ABB RAPID module: dengju.mod

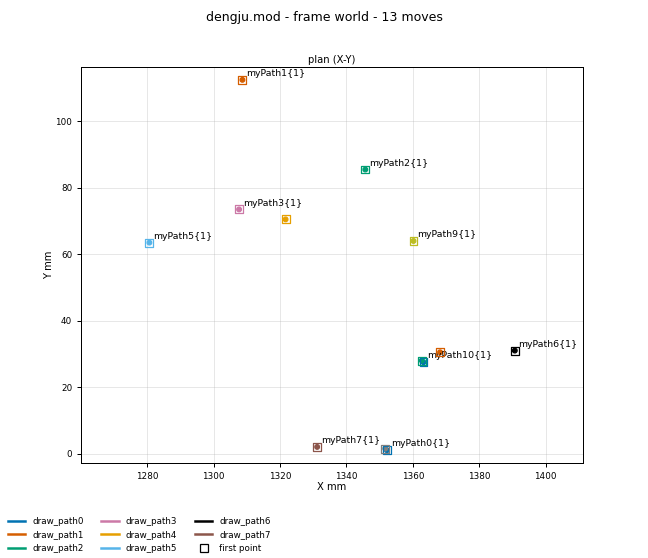
[picture p0: tool path of dengju.mod in frame world, 13 of 26 moves have a stored position in this frame; points joined in program order, loops and branches not executed]
MODULE Module1

    CONST robtarget myPath0{89} := [
        [[1352.2,1,938.01],[0.00139266,-0.491072,0.870802,-0.0234724],[0,-1,-1,0],[9E+09,9E+09,9E+09,9E+09,9E+09,9E+09]],
        [[1347.7,2.5,938.01],[0.00139266,-0.491072,0.870802,-0.0234724],[0,-1,-1,0],[9E+09,9E+09,9E+09,9E+09,9E+09,9E+09]],
        [[1342.2,4.5,938.01],[0.00139266,-0.491072,0.870802,-0.0234724],[0,-1,-1,0],[9E+09,9E+09,9E+09,9E+09,9E+09,9E+09]],
        [[1337.7,2,938.01],[0.00139266,-0.491072,0.870802,-0.0234724],[0,-1,-1,0],[9E+09,9E+09,9E+09,9E+09,9E+09,9E+09]],
        [[1331.7,1.5,938.01],[0.00139266,-0.491072,0.870802,-0.0234724],[0,-1,-1,0],[9E+09,9E+09,9E+09,9E+09,9E+09,9E+09]],
        [[1326.7,2.5,938.01],[0.00139266,-0.491072,0.870802,-0.0234724],[0,-1,-1,0],[9E+09,9E+09,9E+09,9E+09,9E+09,9E+09]],
        [[1322.2,4.5,938.01],[0.00139266,-0.491072,0.870802,-0.0234724],[0,-1,-1,0],[9E+09,9E+09,9E+09,9E+09,9E+09,9E+09]],
        [[1316.2,9.5,938.01],[0.00139266,-0.491072,0.870802,-0.0234724],[0,-1,-1,0],[9E+09,9E+09,9E+09,9E+09,9E+09,9E+09]],
        [[1311.2,14,938.01],[0.00139266,-0.491072,0.870802,-0.0234724],[0,-1,-1,0],[9E+09,9E+09,9E+09,9E+09,9E+09,9E+09]],
        [[1307.2,18,938.01],[0.00139266,-0.491072,0.870802,-0.0234724],[0,-1,-1,0],[9E+09,9E+09,9E+09,9E+09,9E+09,9E+09]],
        [[1304.2,22,938.01],[0.00139266,-0.491072,0.870802,-0.0234724],[0,-1,-1,0],[9E+09,9E+09,9E+09,9E+09,9E+09,9E+09]],
        [[1301.2,26,938.01],[0.00139266,-0.491072,0.870802,-0.0234724],[0,-1,-1,0],[9E+09,9E+09,9E+09,9E+09,9E+09,9E+09]],
        [[1298.7,30,938.01],[0.00139266,-0.491072,0.870802,-0.0234724],[0,-1,-1,0],[9E+09,9E+09,9E+09,9E+09,9E+09,9E+09]],
        [[1296.2,34,938.01],[0.00139266,-0.491072,0.870802,-0.0234724],[0,-1,-1,0],[9E+09,9E+09,9E+09,9E+09,9E+09,9E+09]],
        [[1294.2,38.5,938.01],[0.00139266,-0.491072,0.870802,-0.0234724],[0,-1,-1,0],[9E+09,9E+09,9E+09,9E+09,9E+09,9E+09]],
        [[1292.7,43,938.01],[0.00139266,-0.491072,0.870802,-0.0234724],[0,-1,-1,0],[9E+09,9E+09,9E+09,9E+09,9E+09,9E+09]],
        [[1291.7,51.5,938.01],[0.00139266,-0.491072,0.870802,-0.0234724],[0,-1,-1,0],[9E+09,9E+09,9E+09,9E+09,9E+09,9E+09]],
        [[1293.2,56.5,938.01],[0.00139266,-0.491072,0.870802,-0.0234724],[0,-1,-1,0],[9E+09,9E+09,9E+09,9E+09,9E+09,9E+09]],
        [[1296.7,62,938.01],[0.00139266,-0.491072,0.870802,-0.0234724],[0,-1,-1,0],[9E+09,9E+09,9E+09,9E+09,9E+09,9E+09]],
        [[1300.2,66,938.01],[0.00139266,-0.491072,0.870802,-0.0234724],[0,-1,-1,0],[9E+09,9E+09,9E+09,9E+09,9E+09,9E+09]],
        [[1304.7,69,938.01],[0.00139266,-0.491072,0.870802,-0.0234724],[0,-1,-1,0],[9E+09,9E+09,9E+09,9E+09,9E+09,9E+09]],
        [[1309.2,70.5,938.01],[0.00139266,-0.491072,0.870802,-0.0234724],[0,-1,-1,0],[9E+09,9E+09,9E+09,9E+09,9E+09,9E+09]],
        [[1314.2,71.5,938.01],[0.00139266,-0.491072,0.870802,-0.0234724],[0,-1,-1,0],[9E+09,9E+09,9E+09,9E+09,9E+09,9E+09]],
        [[1318.2,72,938.01],[0.00139266,-0.491072,0.870802,-0.0234724],[0,-1,-1,0],[9E+09,9E+09,9E+09,9E+09,9E+09,9E+09]],
        [[1308.2,73,938.01],[0.00139266,-0.491072,0.870802,-0.0234724],[0,-1,-1,0],[9E+09,9E+09,9E+09,9E+09,9E+09,9E+09]],
        [[1301.2,74,938.01],[0.00139266,-0.491072,0.870802,-0.0234724],[0,-1,-1,0],[9E+09,9E+09,9E+09,9E+09,9E+09,9E+09]],
        [[1296.7,75.5,938.01],[0.00139266,-0.491072,0.870802,-0.0234724],[0,-1,-1,0],[9E+09,9E+09,9E+09,9E+09,9E+09,9E+09]],
        [[1291.7,78,938.01],[0.00139266,-0.491072,0.870802,-0.0234724],[0,-1,-1,0],[9E+09,9E+09,9E+09,9E+09,9E+09,9E+09]],
        [[1287.2,80.5,938.01],[0.00139266,-0.491072,0.870802,-0.0234724],[0,-1,-1,0],[9E+09,9E+09,9E+09,9E+09,9E+09,9E+09]],
        [[1281.7,76.5,938.01],[0.00139266,-0.491072,0.870802,-0.0234724],[0,-1,-1,0],[9E+09,9E+09,9E+09,9E+09,9E+09,9E+09]],
        [[1280.7,69.5,938.01],[0.00139266,-0.491072,0.870802,-0.0234724],[0,-1,-1,0],[9E+09,9E+09,9E+09,9E+09,9E+09,9E+09]],
        [[1283.7,65,938.01],[0.00139266,-0.491072,0.870802,-0.0234724],[0,-1,-1,0],[9E+09,9E+09,9E+09,9E+09,9E+09,9E+09]],
        [[1284.2,63.5,938.01],[0.00139266,-0.491072,0.870802,-0.0234724],[0,-1,-1,0],[9E+09,9E+09,9E+09,9E+09,9E+09,9E+09]],
        [[1279.2,64,938.01],[0.00139266,-0.491072,0.870802,-0.0234724],[0,-1,-1,0],[9E+09,9E+09,9E+09,9E+09,9E+09,9E+09]],
        [[1274.2,66,938.01],[0.00139266,-0.491072,0.870802,-0.0234724],[0,-1,-1,0],[9E+09,9E+09,9E+09,9E+09,9E+09,9E+09]],
        [[1267.2,72,938.01],[0.00139266,-0.491072,0.870802,-0.0234724],[0,-1,-1,0],[9E+09,9E+09,9E+09,9E+09,9E+09,9E+09]],
        [[1265.2,82.5,938.01],[0.00139266,-0.491072,0.870802,-0.0234724],[0,-1,-1,0],[9E+09,9E+09,9E+09,9E+09,9E+09,9E+09]],
        [[1269.2,88,938.01],[0.00139266,-0.491072,0.870802,-0.0234724],[0,-1,-1,0],[9E+09,9E+09,9E+09,9E+09,9E+09,9E+09]],
        [[1274.7,89.5,938.01],[0.00139266,-0.491072,0.870802,-0.0234724],[0,-1,-1,0],[9E+09,9E+09,9E+09,9E+09,9E+09,9E+09]],
        [[1279.7,90.5,938.01],[0.00139266,-0.491072,0.870802,-0.0234724],[0,-1,-1,0],[9E+09,9E+09,9E+09,9E+09,9E+09,9E+09]],
        [[1278.2,98,938.01],[0.00139266,-0.491072,0.870802,-0.0234724],[0,-1,-1,0],[9E+09,9E+09,9E+09,9E+09,9E+09,9E+09]],
        [[1278.2,105.5,938.01],[0.00139266,-0.491072,0.870802,-0.0234724],[0,-1,-1,0],[9E+09,9E+09,9E+09,9E+09,9E+09,9E+09]],
        [[1280.2,110,938.01],[0.00139266,-0.491072,0.870802,-0.0234724],[0,-1,-1,0],[9E+09,9E+09,9E+09,9E+09,9E+09,9E+09]],
        [[1283.7,115.5,938.01],[0.00139266,-0.491072,0.870802,-0.0234724],[0,-1,-1,0],[9E+09,9E+09,9E+09,9E+09,9E+09,9E+09]],
        [[1287.7,119.5,938.01],[0.00139266,-0.491072,0.870802,-0.0234724],[0,-1,-1,0],[9E+09,9E+09,9E+09,9E+09,9E+09,9E+09]],
        [[1293.7,121.5,938.01],[0.00139266,-0.491072,0.870802,-0.0234724],[0,-1,-1,0],[9E+09,9E+09,9E+09,9E+09,9E+09,9E+09]],
        [[1301.2,121.5,938.01],[0.00139266,-0.491072,0.870802,-0.0234724],[0,-1,-1,0],[9E+09,9E+09,9E+09,9E+09,9E+09,9E+09]],
        [[1305.7,120,938.01],[0.00139266,-0.491072,0.870802,-0.0234724],[0,-1,-1,0],[9E+09,9E+09,9E+09,9E+09,9E+09,9E+09]],
        [[1310.7,119,938.01],[0.00139266,-0.491072,0.870802,-0.0234724],[0,-1,-1,0],[9E+09,9E+09,9E+09,9E+09,9E+09,9E+09]],
        [[1311.7,115,938.01],[0.00139266,-0.491072,0.870802,-0.0234724],[0,-1,-1,0],[9E+09,9E+09,9E+09,9E+09,9E+09,9E+09]],
        [[1320.2,114,938.01],[0.00139266,-0.491072,0.870802,-0.0234724],[0,-1,-1,0],[9E+09,9E+09,9E+09,9E+09,9E+09,9E+09]],
        [[1324.7,120,938.01],[0.00139266,-0.491072,0.870802,-0.0234724],[0,-1,-1,0],[9E+09,9E+09,9E+09,9E+09,9E+09,9E+09]],
        [[1331.7,121.5,938.01],[0.00139266,-0.491072,0.870802,-0.0234724],[0,-1,-1,0],[9E+09,9E+09,9E+09,9E+09,9E+09,9E+09]],
        [[1337.7,122,938.01],[0.00139266,-0.491072,0.870802,-0.0234724],[0,-1,-1,0],[9E+09,9E+09,9E+09,9E+09,9E+09,9E+09]],
        [[1342.7,121,938.01],[0.00139266,-0.491072,0.870802,-0.0234724],[0,-1,-1,0],[9E+09,9E+09,9E+09,9E+09,9E+09,9E+09]],
        [[1345.7,116,938.01],[0.00139266,-0.491072,0.870802,-0.0234724],[0,-1,-1,0],[9E+09,9E+09,9E+09,9E+09,9E+09,9E+09]],
        [[1346.7,113,938.01],[0.00139266,-0.491072,0.870802,-0.0234724],[0,-1,-1,0],[9E+09,9E+09,9E+09,9E+09,9E+09,9E+09]],
        [[1351.2,111.5,938.01],[0.00139266,-0.491072,0.870802,-0.0234724],[0,-1,-1,0],[9E+09,9E+09,9E+09,9E+09,9E+09,9E+09]],
        [[1356.7,108,938.01],[0.00139266,-0.491072,0.870802,-0.0234724],[0,-1,-1,0],[9E+09,9E+09,9E+09,9E+09,9E+09,9E+09]],
        [[1354.7,103.5,938.01],[0.00139266,-0.491072,0.870802,-0.0234724],[0,-1,-1,0],[9E+09,9E+09,9E+09,9E+09,9E+09,9E+09]],
        [[1352.7,99,938.01],[0.00139266,-0.491072,0.870802,-0.0234724],[0,-1,-1,0],[9E+09,9E+09,9E+09,9E+09,9E+09,9E+09]],
        [[1351.2,94,938.01],[0.00139266,-0.491072,0.870802,-0.0234724],[0,-1,-1,0],[9E+09,9E+09,9E+09,9E+09,9E+09,9E+09]],
        [[1352.2,89,938.01],[0.00139266,-0.491072,0.870802,-0.0234724],[0,-1,-1,0],[9E+09,9E+09,9E+09,9E+09,9E+09,9E+09]],
        [[1351.7,85,938.01],[0.00139266,-0.491072,0.870802,-0.0234724],[0,-1,-1,0],[9E+09,9E+09,9E+09,9E+09,9E+09,9E+09]],
        [[1354.2,80.5,938.01],[0.00139266,-0.491072,0.870802,-0.0234724],[0,-1,-1,0],[9E+09,9E+09,9E+09,9E+09,9E+09,9E+09]],
        [[1361.2,80,938.01],[0.00139266,-0.491072,0.870802,-0.0234724],[0,-1,-1,0],[9E+09,9E+09,9E+09,9E+09,9E+09,9E+09]],
        [[1366.2,79,938.01],[0.00139266,-0.491072,0.870802,-0.0234724],[0,-1,-1,0],[9E+09,9E+09,9E+09,9E+09,9E+09,9E+09]],
        [[1371.2,77.5,938.01],[0.00139266,-0.491072,0.870802,-0.0234724],[0,-1,-1,0],[9E+09,9E+09,9E+09,9E+09,9E+09,9E+09]],
        [[1375.7,75.5,938.01],[0.00139266,-0.491072,0.870802,-0.0234724],[0,-1,-1,0],[9E+09,9E+09,9E+09,9E+09,9E+09,9E+09]],
        [[1380.2,73.5,938.01],[0.00139266,-0.491072,0.870802,-0.0234724],[0,-1,-1,0],[9E+09,9E+09,9E+09,9E+09,9E+09,9E+09]],
        [[1384.2,71,938.01],[0.00139266,-0.491072,0.870802,-0.0234724],[0,-1,-1,0],[9E+09,9E+09,9E+09,9E+09,9E+09,9E+09]],
        [[1388.2,68.5,938.01],[0.00139266,-0.491072,0.870802,-0.0234724],[0,-1,-1,0],[9E+09,9E+09,9E+09,9E+09,9E+09,9E+09]],
        [[1393.2,63.5,938.01],[0.00139266,-0.491072,0.870802,-0.0234724],[0,-1,-1,0],[9E+09,9E+09,9E+09,9E+09,9E+09,9E+09]],
        [[1395.7,59,938.01],[0.00139266,-0.491072,0.870802,-0.0234724],[0,-1,-1,0],[9E+09,9E+09,9E+09,9E+09,9E+09,9E+09]],
        [[1398.2,55,938.01],[0.00139266,-0.491072,0.870802,-0.0234724],[0,-1,-1,0],[9E+09,9E+09,9E+09,9E+09,9E+09,9E+09]],
        [[1398.7,49.5,938.01],[0.00139266,-0.491072,0.870802,-0.0234724],[0,-1,-1,0],[9E+09,9E+09,9E+09,9E+09,9E+09,9E+09]],
        [[1397.7,44.5,938.01],[0.00139266,-0.491072,0.870802,-0.0234724],[0,-1,-1,0],[9E+09,9E+09,9E+09,9E+09,9E+09,9E+09]],
        [[1401.2,41.5,938.01],[0.00139266,-0.491072,0.870802,-0.0234724],[0,-1,-1,0],[9E+09,9E+09,9E+09,9E+09,9E+09,9E+09]],
        [[1401.7,36,938.01],[0.00139266,-0.491072,0.870802,-0.0234724],[0,-1,-1,0],[9E+09,9E+09,9E+09,9E+09,9E+09,9E+09]],
        [[1397.7,32,938.01],[0.00139266,-0.491072,0.870802,-0.0234724],[0,-1,-1,0],[9E+09,9E+09,9E+09,9E+09,9E+09,9E+09]],
        [[1392.7,31,938.01],[0.00139266,-0.491072,0.870802,-0.0234724],[0,-1,-1,0],[9E+09,9E+09,9E+09,9E+09,9E+09,9E+09]],
        [[1385.7,26,938.01],[0.00139266,-0.491072,0.870802,-0.0234724],[0,-1,-1,0],[9E+09,9E+09,9E+09,9E+09,9E+09,9E+09]],
        [[1382.7,22,938.01],[0.00139266,-0.491072,0.870802,-0.0234724],[0,-1,-1,0],[9E+09,9E+09,9E+09,9E+09,9E+09,9E+09]],
        [[1380.2,18,938.01],[0.00139266,-0.491072,0.870802,-0.0234724],[0,-1,-1,0],[9E+09,9E+09,9E+09,9E+09,9E+09,9E+09]],
        [[1375.7,12.5,938.01],[0.00139266,-0.491072,0.870802,-0.0234724],[0,-1,-1,0],[9E+09,9E+09,9E+09,9E+09,9E+09,9E+09]],
        [[1371.2,7.5,938.01],[0.00139266,-0.491072,0.870802,-0.0234724],[0,-1,-1,0],[9E+09,9E+09,9E+09,9E+09,9E+09,9E+09]],
        [[1367.2,5,938.01],[0.00139266,-0.491072,0.870802,-0.0234724],[0,-1,-1,0],[9E+09,9E+09,9E+09,9E+09,9E+09,9E+09]],
        [[1362.7,2.5,938.01],[0.00139266,-0.491072,0.870802,-0.0234724],[0,-1,-1,0],[9E+09,9E+09,9E+09,9E+09,9E+09,9E+09]],
        [[1357.7,1.5,938.01],[0.00139266,-0.491072,0.870802,-0.0234724],[0,-1,-1,0],[9E+09,9E+09,9E+09,9E+09,9E+09,9E+09]]
        ];
    CONST robtarget myPath1{4} := [
        [[1308.7,112.5,938.01],[0.00139266,-0.491072,0.870802,-0.0234724],[0,-1,-1,0],[9E+09,9E+09,9E+09,9E+09,9E+09,9E+09]],
        [[1312.2,115.5,938.01],[0.00139266,-0.491072,0.870802,-0.0234724],[0,-1,-1,0],[9E+09,9E+09,9E+09,9E+09,9E+09,9E+09]],
        [[1310.2,119,938.01],[0.00139266,-0.491072,0.870802,-0.0234724],[0,-1,-1,0],[9E+09,9E+09,9E+09,9E+09,9E+09,9E+09]],
        [[1306.2,116.5,938.01],[0.00139266,-0.491072,0.870802,-0.0234724],[0,-1,-1,0],[9E+09,9E+09,9E+09,9E+09,9E+09,9E+09]]
        ];
    CONST robtarget myPath2{5} := [
        [[1345.7,85.5,938.01],[0.00139266,-0.491072,0.870802,-0.0234724],[0,-1,-1,0],[9E+09,9E+09,9E+09,9E+09,9E+09,9E+09]],
        [[1350.7,86.5,938.01],[0.00139266,-0.491072,0.870802,-0.0234724],[0,-1,-1,0],[9E+09,9E+09,9E+09,9E+09,9E+09,9E+09]],
        [[1352.2,93,938.01],[0.00139266,-0.491072,0.870802,-0.0234724],[0,-1,-1,0],[9E+09,9E+09,9E+09,9E+09,9E+09,9E+09]],
        [[1348.2,95.5,938.01],[0.00139266,-0.491072,0.870802,-0.0234724],[0,-1,-1,0],[9E+09,9E+09,9E+09,9E+09,9E+09,9E+09]],
        [[1342.2,92.5,938.01],[0.00139266,-0.491072,0.870802,-0.0234724],[0,-1,-1,0],[9E+09,9E+09,9E+09,9E+09,9E+09,9E+09]]
        ];
    CONST robtarget myPath3{54} := [
        [[1307.7,73.5,938.01],[0.00139266,-0.491072,0.870802,-0.0234724],[0,-1,-1,0],[9E+09,9E+09,9E+09,9E+09,9E+09,9E+09]],
        [[1317.2,73,938.01],[0.00139266,-0.491072,0.870802,-0.0234724],[0,-1,-1,0],[9E+09,9E+09,9E+09,9E+09,9E+09,9E+09]],
        [[1319.7,77,938.01],[0.00139266,-0.491072,0.870802,-0.0234724],[0,-1,-1,0],[9E+09,9E+09,9E+09,9E+09,9E+09,9E+09]],
        [[1323.7,82,938.01],[0.00139266,-0.491072,0.870802,-0.0234724],[0,-1,-1,0],[9E+09,9E+09,9E+09,9E+09,9E+09,9E+09]],
        [[1327.7,84.5,938.01],[0.00139266,-0.491072,0.870802,-0.0234724],[0,-1,-1,0],[9E+09,9E+09,9E+09,9E+09,9E+09,9E+09]],
        [[1332.7,87,938.01],[0.00139266,-0.491072,0.870802,-0.0234724],[0,-1,-1,0],[9E+09,9E+09,9E+09,9E+09,9E+09,9E+09]],
        [[1337.2,88.5,938.01],[0.00139266,-0.491072,0.870802,-0.0234724],[0,-1,-1,0],[9E+09,9E+09,9E+09,9E+09,9E+09,9E+09]],
        [[1342.2,89.5,938.01],[0.00139266,-0.491072,0.870802,-0.0234724],[0,-1,-1,0],[9E+09,9E+09,9E+09,9E+09,9E+09,9E+09]],
        [[1344.7,95,938.01],[0.00139266,-0.491072,0.870802,-0.0234724],[0,-1,-1,0],[9E+09,9E+09,9E+09,9E+09,9E+09,9E+09]],
        [[1350.7,95,938.01],[0.00139266,-0.491072,0.870802,-0.0234724],[0,-1,-1,0],[9E+09,9E+09,9E+09,9E+09,9E+09,9E+09]],
        [[1352.7,101,938.01],[0.00139266,-0.491072,0.870802,-0.0234724],[0,-1,-1,0],[9E+09,9E+09,9E+09,9E+09,9E+09,9E+09]],
        [[1356.7,105.5,938.01],[0.00139266,-0.491072,0.870802,-0.0234724],[0,-1,-1,0],[9E+09,9E+09,9E+09,9E+09,9E+09,9E+09]],
        [[1354.2,110.5,938.01],[0.00139266,-0.491072,0.870802,-0.0234724],[0,-1,-1,0],[9E+09,9E+09,9E+09,9E+09,9E+09,9E+09]],
        [[1349.2,112,938.01],[0.00139266,-0.491072,0.870802,-0.0234724],[0,-1,-1,0],[9E+09,9E+09,9E+09,9E+09,9E+09,9E+09]],
        [[1344.7,113.5,938.01],[0.00139266,-0.491072,0.870802,-0.0234724],[0,-1,-1,0],[9E+09,9E+09,9E+09,9E+09,9E+09,9E+09]],
        [[1342.7,107.5,938.01],[0.00139266,-0.491072,0.870802,-0.0234724],[0,-1,-1,0],[9E+09,9E+09,9E+09,9E+09,9E+09,9E+09]],
        [[1343.7,103.5,938.01],[0.00139266,-0.491072,0.870802,-0.0234724],[0,-1,-1,0],[9E+09,9E+09,9E+09,9E+09,9E+09,9E+09]],
        [[1343.7,103.5,938.01],[0.00139266,-0.491072,0.870802,-0.0234724],[0,-1,-1,0],[9E+09,9E+09,9E+09,9E+09,9E+09,9E+09]],
        [[1340.2,101,938.01],[0.00139266,-0.491072,0.870802,-0.0234724],[0,-1,-1,0],[9E+09,9E+09,9E+09,9E+09,9E+09,9E+09]],
        [[1341.7,104,938.01],[0.00139266,-0.491072,0.870802,-0.0234724],[0,-1,-1,0],[9E+09,9E+09,9E+09,9E+09,9E+09,9E+09]],
        [[1342.7,111,938.01],[0.00139266,-0.491072,0.870802,-0.0234724],[0,-1,-1,0],[9E+09,9E+09,9E+09,9E+09,9E+09,9E+09]],
        [[1344.7,115,938.01],[0.00139266,-0.491072,0.870802,-0.0234724],[0,-1,-1,0],[9E+09,9E+09,9E+09,9E+09,9E+09,9E+09]],
        [[1343.7,120.5,938.01],[0.00139266,-0.491072,0.870802,-0.0234724],[0,-1,-1,0],[9E+09,9E+09,9E+09,9E+09,9E+09,9E+09]],
        [[1338.2,121.5,938.01],[0.00139266,-0.491072,0.870802,-0.0234724],[0,-1,-1,0],[9E+09,9E+09,9E+09,9E+09,9E+09,9E+09]],
        [[1332.2,122,938.01],[0.00139266,-0.491072,0.870802,-0.0234724],[0,-1,-1,0],[9E+09,9E+09,9E+09,9E+09,9E+09,9E+09]],
        [[1327.2,121,938.01],[0.00139266,-0.491072,0.870802,-0.0234724],[0,-1,-1,0],[9E+09,9E+09,9E+09,9E+09,9E+09,9E+09]],
        [[1323.2,118,938.01],[0.00139266,-0.491072,0.870802,-0.0234724],[0,-1,-1,0],[9E+09,9E+09,9E+09,9E+09,9E+09,9E+09]],
        [[1320.7,114,938.01],[0.00139266,-0.491072,0.870802,-0.0234724],[0,-1,-1,0],[9E+09,9E+09,9E+09,9E+09,9E+09,9E+09]],
        [[1320.2,113.5,938.01],[0.00139266,-0.491072,0.870802,-0.0234724],[0,-1,-1,0],[9E+09,9E+09,9E+09,9E+09,9E+09,9E+09]],
        [[1314.2,114,938.01],[0.00139266,-0.491072,0.870802,-0.0234724],[0,-1,-1,0],[9E+09,9E+09,9E+09,9E+09,9E+09,9E+09]],
        [[1309.7,112.5,938.01],[0.00139266,-0.491072,0.870802,-0.0234724],[0,-1,-1,0],[9E+09,9E+09,9E+09,9E+09,9E+09,9E+09]],
        [[1309.2,106,938.01],[0.00139266,-0.491072,0.870802,-0.0234724],[0,-1,-1,0],[9E+09,9E+09,9E+09,9E+09,9E+09,9E+09]],
        [[1309.2,101,938.01],[0.00139266,-0.491072,0.870802,-0.0234724],[0,-1,-1,0],[9E+09,9E+09,9E+09,9E+09,9E+09,9E+09]],
        [[1306.7,96,938.01],[0.00139266,-0.491072,0.870802,-0.0234724],[0,-1,-1,0],[9E+09,9E+09,9E+09,9E+09,9E+09,9E+09]],
        [[1308.2,98,938.01],[0.00139266,-0.491072,0.870802,-0.0234724],[0,-1,-1,0],[9E+09,9E+09,9E+09,9E+09,9E+09,9E+09]],
        [[1309.2,104,938.01],[0.00139266,-0.491072,0.870802,-0.0234724],[0,-1,-1,0],[9E+09,9E+09,9E+09,9E+09,9E+09,9E+09]],
        [[1309.2,109.5,938.01],[0.00139266,-0.491072,0.870802,-0.0234724],[0,-1,-1,0],[9E+09,9E+09,9E+09,9E+09,9E+09,9E+09]],
        [[1307.7,114,938.01],[0.00139266,-0.491072,0.870802,-0.0234724],[0,-1,-1,0],[9E+09,9E+09,9E+09,9E+09,9E+09,9E+09]],
        [[1306.2,119,938.01],[0.00139266,-0.491072,0.870802,-0.0234724],[0,-1,-1,0],[9E+09,9E+09,9E+09,9E+09,9E+09,9E+09]],
        [[1301.7,121,938.01],[0.00139266,-0.491072,0.870802,-0.0234724],[0,-1,-1,0],[9E+09,9E+09,9E+09,9E+09,9E+09,9E+09]],
        [[1294.2,122,938.01],[0.00139266,-0.491072,0.870802,-0.0234724],[0,-1,-1,0],[9E+09,9E+09,9E+09,9E+09,9E+09,9E+09]],
        [[1289.7,120.5,938.01],[0.00139266,-0.491072,0.870802,-0.0234724],[0,-1,-1,0],[9E+09,9E+09,9E+09,9E+09,9E+09,9E+09]],
        [[1285.7,117.5,938.01],[0.00139266,-0.491072,0.870802,-0.0234724],[0,-1,-1,0],[9E+09,9E+09,9E+09,9E+09,9E+09,9E+09]],
        [[1281.7,113.5,938.01],[0.00139266,-0.491072,0.870802,-0.0234724],[0,-1,-1,0],[9E+09,9E+09,9E+09,9E+09,9E+09,9E+09]],
        [[1279.7,109,938.01],[0.00139266,-0.491072,0.870802,-0.0234724],[0,-1,-1,0],[9E+09,9E+09,9E+09,9E+09,9E+09,9E+09]],
        [[1278.2,102.5,938.01],[0.00139266,-0.491072,0.870802,-0.0234724],[0,-1,-1,0],[9E+09,9E+09,9E+09,9E+09,9E+09,9E+09]],
        [[1278.2,94.5,938.01],[0.00139266,-0.491072,0.870802,-0.0234724],[0,-1,-1,0],[9E+09,9E+09,9E+09,9E+09,9E+09,9E+09]],
        [[1279.7,90,938.01],[0.00139266,-0.491072,0.870802,-0.0234724],[0,-1,-1,0],[9E+09,9E+09,9E+09,9E+09,9E+09,9E+09]],
        [[1282.2,86,938.01],[0.00139266,-0.491072,0.870802,-0.0234724],[0,-1,-1,0],[9E+09,9E+09,9E+09,9E+09,9E+09,9E+09]],
        [[1286.2,81.5,938.01],[0.00139266,-0.491072,0.870802,-0.0234724],[0,-1,-1,0],[9E+09,9E+09,9E+09,9E+09,9E+09,9E+09]],
        [[1290.2,78.5,938.01],[0.00139266,-0.491072,0.870802,-0.0234724],[0,-1,-1,0],[9E+09,9E+09,9E+09,9E+09,9E+09,9E+09]],
        [[1295.2,76,938.01],[0.00139266,-0.491072,0.870802,-0.0234724],[0,-1,-1,0],[9E+09,9E+09,9E+09,9E+09,9E+09,9E+09]],
        [[1299.7,74.5,938.01],[0.00139266,-0.491072,0.870802,-0.0234724],[0,-1,-1,0],[9E+09,9E+09,9E+09,9E+09,9E+09,9E+09]],
        [[1304.7,73.5,938.01],[0.00139266,-0.491072,0.870802,-0.0234724],[0,-1,-1,0],[9E+09,9E+09,9E+09,9E+09,9E+09,9E+09]]
        ];
    CONST robtarget myPath4{15} := [
        [[1321.7,70.5,938.01],[0.00139266,-0.491072,0.870802,-0.0234724],[0,-1,-1,0],[9E+09,9E+09,9E+09,9E+09,9E+09,9E+09]],
        [[1328.7,75,938.01],[0.00139266,-0.491072,0.870802,-0.0234724],[0,-1,-1,0],[9E+09,9E+09,9E+09,9E+09,9E+09,9E+09]],
        [[1333.2,77.5,938.01],[0.00139266,-0.491072,0.870802,-0.0234724],[0,-1,-1,0],[9E+09,9E+09,9E+09,9E+09,9E+09,9E+09]],
        [[1338.2,79,938.01],[0.00139266,-0.491072,0.870802,-0.0234724],[0,-1,-1,0],[9E+09,9E+09,9E+09,9E+09,9E+09,9E+09]],
        [[1343.7,80,938.01],[0.00139266,-0.491072,0.870802,-0.0234724],[0,-1,-1,0],[9E+09,9E+09,9E+09,9E+09,9E+09,9E+09]],
        [[1352.7,80.5,938.01],[0.00139266,-0.491072,0.870802,-0.0234724],[0,-1,-1,0],[9E+09,9E+09,9E+09,9E+09,9E+09,9E+09]],
        [[1350.7,86,938.01],[0.00139266,-0.491072,0.870802,-0.0234724],[0,-1,-1,0],[9E+09,9E+09,9E+09,9E+09,9E+09,9E+09]],
        [[1345.7,85.5,938.01],[0.00139266,-0.491072,0.870802,-0.0234724],[0,-1,-1,0],[9E+09,9E+09,9E+09,9E+09,9E+09,9E+09]],
        [[1342.2,88.5,938.01],[0.00139266,-0.491072,0.870802,-0.0234724],[0,-1,-1,0],[9E+09,9E+09,9E+09,9E+09,9E+09,9E+09]],
        [[1337.2,88.5,938.01],[0.00139266,-0.491072,0.870802,-0.0234724],[0,-1,-1,0],[9E+09,9E+09,9E+09,9E+09,9E+09,9E+09]],
        [[1332.7,86.5,938.01],[0.00139266,-0.491072,0.870802,-0.0234724],[0,-1,-1,0],[9E+09,9E+09,9E+09,9E+09,9E+09,9E+09]],
        [[1328.2,84.5,938.01],[0.00139266,-0.491072,0.870802,-0.0234724],[0,-1,-1,0],[9E+09,9E+09,9E+09,9E+09,9E+09,9E+09]],
        [[1323.2,81,938.01],[0.00139266,-0.491072,0.870802,-0.0234724],[0,-1,-1,0],[9E+09,9E+09,9E+09,9E+09,9E+09,9E+09]],
        [[1319.7,77.5,938.01],[0.00139266,-0.491072,0.870802,-0.0234724],[0,-1,-1,0],[9E+09,9E+09,9E+09,9E+09,9E+09,9E+09]],
        [[1318.2,72,938.01],[0.00139266,-0.491072,0.870802,-0.0234724],[0,-1,-1,0],[9E+09,9E+09,9E+09,9E+09,9E+09,9E+09]]
        ];
    CONST robtarget myPath5{15} := [
        [[1280.7,63.5,938.01],[0.00139266,-0.491072,0.870802,-0.0234724],[0,-1,-1,0],[9E+09,9E+09,9E+09,9E+09,9E+09,9E+09]],
        [[1283.7,65,938.01],[0.00139266,-0.491072,0.870802,-0.0234724],[0,-1,-1,0],[9E+09,9E+09,9E+09,9E+09,9E+09,9E+09]],
        [[1281.2,69,938.01],[0.00139266,-0.491072,0.870802,-0.0234724],[0,-1,-1,0],[9E+09,9E+09,9E+09,9E+09,9E+09,9E+09]],
        [[1280.7,74.5,938.01],[0.00139266,-0.491072,0.870802,-0.0234724],[0,-1,-1,0],[9E+09,9E+09,9E+09,9E+09,9E+09,9E+09]],
        [[1284.7,79.5,938.01],[0.00139266,-0.491072,0.870802,-0.0234724],[0,-1,-1,0],[9E+09,9E+09,9E+09,9E+09,9E+09,9E+09]],
        [[1285.2,82.5,938.01],[0.00139266,-0.491072,0.870802,-0.0234724],[0,-1,-1,0],[9E+09,9E+09,9E+09,9E+09,9E+09,9E+09]],
        [[1282.2,86,938.01],[0.00139266,-0.491072,0.870802,-0.0234724],[0,-1,-1,0],[9E+09,9E+09,9E+09,9E+09,9E+09,9E+09]],
        [[1279.7,90,938.01],[0.00139266,-0.491072,0.870802,-0.0234724],[0,-1,-1,0],[9E+09,9E+09,9E+09,9E+09,9E+09,9E+09]],
        [[1273.2,89.5,938.01],[0.00139266,-0.491072,0.870802,-0.0234724],[0,-1,-1,0],[9E+09,9E+09,9E+09,9E+09,9E+09,9E+09]],
        [[1268.7,87.5,938.01],[0.00139266,-0.491072,0.870802,-0.0234724],[0,-1,-1,0],[9E+09,9E+09,9E+09,9E+09,9E+09,9E+09]],
        [[1265.7,83.5,938.01],[0.00139266,-0.491072,0.870802,-0.0234724],[0,-1,-1,0],[9E+09,9E+09,9E+09,9E+09,9E+09,9E+09]],
        [[1265.2,76.5,938.01],[0.00139266,-0.491072,0.870802,-0.0234724],[0,-1,-1,0],[9E+09,9E+09,9E+09,9E+09,9E+09,9E+09]],
        [[1267.2,72,938.01],[0.00139266,-0.491072,0.870802,-0.0234724],[0,-1,-1,0],[9E+09,9E+09,9E+09,9E+09,9E+09,9E+09]],
        [[1272.2,67,938.01],[0.00139266,-0.491072,0.870802,-0.0234724],[0,-1,-1,0],[9E+09,9E+09,9E+09,9E+09,9E+09,9E+09]],
        [[1276.2,64.5,938.01],[0.00139266,-0.491072,0.870802,-0.0234724],[0,-1,-1,0],[9E+09,9E+09,9E+09,9E+09,9E+09,9E+09]]
        ];
    CONST robtarget myPath6{8} := [
        [[1390.7,31,938.01],[0.00139266,-0.491072,0.870802,-0.0234724],[0,-1,-1,0],[9E+09,9E+09,9E+09,9E+09,9E+09,9E+09]],
        [[1395.7,31.5,938.01],[0.00139266,-0.491072,0.870802,-0.0234724],[0,-1,-1,0],[9E+09,9E+09,9E+09,9E+09,9E+09,9E+09]],
        [[1400.7,34.5,938.01],[0.00139266,-0.491072,0.870802,-0.0234724],[0,-1,-1,0],[9E+09,9E+09,9E+09,9E+09,9E+09,9E+09]],
        [[1401.7,40.5,938.01],[0.00139266,-0.491072,0.870802,-0.0234724],[0,-1,-1,0],[9E+09,9E+09,9E+09,9E+09,9E+09,9E+09]],
        [[1398.2,44,938.01],[0.00139266,-0.491072,0.870802,-0.0234724],[0,-1,-1,0],[9E+09,9E+09,9E+09,9E+09,9E+09,9E+09]],
        [[1393.2,43,938.01],[0.00139266,-0.491072,0.870802,-0.0234724],[0,-1,-1,0],[9E+09,9E+09,9E+09,9E+09,9E+09,9E+09]],
        [[1388.2,39.5,938.01],[0.00139266,-0.491072,0.870802,-0.0234724],[0,-1,-1,0],[9E+09,9E+09,9E+09,9E+09,9E+09,9E+09]],
        [[1387.7,34.5,938.01],[0.00139266,-0.491072,0.870802,-0.0234724],[0,-1,-1,0],[9E+09,9E+09,9E+09,9E+09,9E+09,9E+09]]
        ];
    CONST robtarget myPath7{36} := [
        [[1331.2,2,938.01],[0.00139266,-0.491072,0.870802,-0.0234724],[0,-1,-1,0],[9E+09,9E+09,9E+09,9E+09,9E+09,9E+09]],
        [[1336.2,2,938.01],[0.00139266,-0.491072,0.870802,-0.0234724],[0,-1,-1,0],[9E+09,9E+09,9E+09,9E+09,9E+09,9E+09]],
        [[1340.7,3.5,938.01],[0.00139266,-0.491072,0.870802,-0.0234724],[0,-1,-1,0],[9E+09,9E+09,9E+09,9E+09,9E+09,9E+09]],
        [[1343.7,7,938.01],[0.00139266,-0.491072,0.870802,-0.0234724],[0,-1,-1,0],[9E+09,9E+09,9E+09,9E+09,9E+09,9E+09]],
        [[1345.7,12.5,938.01],[0.00139266,-0.491072,0.870802,-0.0234724],[0,-1,-1,0],[9E+09,9E+09,9E+09,9E+09,9E+09,9E+09]],
        [[1346.2,18.5,938.01],[0.00139266,-0.491072,0.870802,-0.0234724],[0,-1,-1,0],[9E+09,9E+09,9E+09,9E+09,9E+09,9E+09]],
        [[1345.2,24.5,938.01],[0.00139266,-0.491072,0.870802,-0.0234724],[0,-1,-1,0],[9E+09,9E+09,9E+09,9E+09,9E+09,9E+09]],
        [[1343.7,29,938.01],[0.00139266,-0.491072,0.870802,-0.0234724],[0,-1,-1,0],[9E+09,9E+09,9E+09,9E+09,9E+09,9E+09]],
        [[1342.7,35.5,938.01],[0.00139266,-0.491072,0.870802,-0.0234724],[0,-1,-1,0],[9E+09,9E+09,9E+09,9E+09,9E+09,9E+09]],
        [[1341.2,40,938.01],[0.00139266,-0.491072,0.870802,-0.0234724],[0,-1,-1,0],[9E+09,9E+09,9E+09,9E+09,9E+09,9E+09]],
        [[1340.2,45.5,938.01],[0.00139266,-0.491072,0.870802,-0.0234724],[0,-1,-1,0],[9E+09,9E+09,9E+09,9E+09,9E+09,9E+09]],
        [[1338.2,50,938.01],[0.00139266,-0.491072,0.870802,-0.0234724],[0,-1,-1,0],[9E+09,9E+09,9E+09,9E+09,9E+09,9E+09]],
        [[1336.7,54.5,938.01],[0.00139266,-0.491072,0.870802,-0.0234724],[0,-1,-1,0],[9E+09,9E+09,9E+09,9E+09,9E+09,9E+09]],
        [[1334.2,59,938.01],[0.00139266,-0.491072,0.870802,-0.0234724],[0,-1,-1,0],[9E+09,9E+09,9E+09,9E+09,9E+09,9E+09]],
        [[1331.7,63,938.01],[0.00139266,-0.491072,0.870802,-0.0234724],[0,-1,-1,0],[9E+09,9E+09,9E+09,9E+09,9E+09,9E+09]],
        [[1328.2,67,938.01],[0.00139266,-0.491072,0.870802,-0.0234724],[0,-1,-1,0],[9E+09,9E+09,9E+09,9E+09,9E+09,9E+09]],
        [[1323.7,70,938.01],[0.00139266,-0.491072,0.870802,-0.0234724],[0,-1,-1,0],[9E+09,9E+09,9E+09,9E+09,9E+09,9E+09]],
        [[1318.7,71.5,938.01],[0.00139266,-0.491072,0.870802,-0.0234724],[0,-1,-1,0],[9E+09,9E+09,9E+09,9E+09,9E+09,9E+09]],
        [[1314.2,71,938.01],[0.00139266,-0.491072,0.870802,-0.0234724],[0,-1,-1,0],[9E+09,9E+09,9E+09,9E+09,9E+09,9E+09]],
        [[1309.2,70.5,938.01],[0.00139266,-0.491072,0.870802,-0.0234724],[0,-1,-1,0],[9E+09,9E+09,9E+09,9E+09,9E+09,9E+09]],
        [[1304.7,69,938.01],[0.00139266,-0.491072,0.870802,-0.0234724],[0,-1,-1,0],[9E+09,9E+09,9E+09,9E+09,9E+09,9E+09]],
        [[1300.2,65.5,938.01],[0.00139266,-0.491072,0.870802,-0.0234724],[0,-1,-1,0],[9E+09,9E+09,9E+09,9E+09,9E+09,9E+09]],
        [[1296.7,62,938.01],[0.00139266,-0.491072,0.870802,-0.0234724],[0,-1,-1,0],[9E+09,9E+09,9E+09,9E+09,9E+09,9E+09]],
        [[1293.7,58,938.01],[0.00139266,-0.491072,0.870802,-0.0234724],[0,-1,-1,0],[9E+09,9E+09,9E+09,9E+09,9E+09,9E+09]],
        [[1292.2,52,938.01],[0.00139266,-0.491072,0.870802,-0.0234724],[0,-1,-1,0],[9E+09,9E+09,9E+09,9E+09,9E+09,9E+09]],
        [[1291.7,47,938.01],[0.00139266,-0.491072,0.870802,-0.0234724],[0,-1,-1,0],[9E+09,9E+09,9E+09,9E+09,9E+09,9E+09]],
        [[1293.2,42,938.01],[0.00139266,-0.491072,0.870802,-0.0234724],[0,-1,-1,0],[9E+09,9E+09,9E+09,9E+09,9E+09,9E+09]],
        [[1294.7,37,938.01],[0.00139266,-0.491072,0.870802,-0.0234724],[0,-1,-1,0],[9E+09,9E+09,9E+09,9E+09,9E+09,9E+09]],
        [[1297.2,33,938.01],[0.00139266,-0.491072,0.870802,-0.0234724],[0,-1,-1,0],[9E+09,9E+09,9E+09,9E+09,9E+09,9E+09]],
        [[1299.7,29,938.01],[0.00139266,-0.491072,0.870802,-0.0234724],[0,-1,-1,0],[9E+09,9E+09,9E+09,9E+09,9E+09,9E+09]],
        [[1302.7,24.5,938.01],[0.00139266,-0.491072,0.870802,-0.0234724],[0,-1,-1,0],[9E+09,9E+09,9E+09,9E+09,9E+09,9E+09]],
        [[1307.2,18.5,938.01],[0.00139266,-0.491072,0.870802,-0.0234724],[0,-1,-1,0],[9E+09,9E+09,9E+09,9E+09,9E+09,9E+09]],
        [[1314.7,10.5,938.01],[0.00139266,-0.491072,0.870802,-0.0234724],[0,-1,-1,0],[9E+09,9E+09,9E+09,9E+09,9E+09,9E+09]],
        [[1318.2,7.5,938.01],[0.00139266,-0.491072,0.870802,-0.0234724],[0,-1,-1,0],[9E+09,9E+09,9E+09,9E+09,9E+09,9E+09]],
        [[1323.2,4,938.01],[0.00139266,-0.491072,0.870802,-0.0234724],[0,-1,-1,0],[9E+09,9E+09,9E+09,9E+09,9E+09,9E+09]],
        [[1328.2,2.5,938.01],[0.00139266,-0.491072,0.870802,-0.0234724],[0,-1,-1,0],[9E+09,9E+09,9E+09,9E+09,9E+09,9E+09]]
        ];
    CONST robtarget myPath8{46} := [
        [[1351.7,1.5,938.01],[0.00139266,-0.491072,0.870802,-0.0234724],[0,-1,-1,0],[9E+09,9E+09,9E+09,9E+09,9E+09,9E+09]],
        [[1357.2,1,938.01],[0.00139266,-0.491072,0.870802,-0.0234724],[0,-1,-1,0],[9E+09,9E+09,9E+09,9E+09,9E+09,9E+09]],
        [[1362.2,2.5,938.01],[0.00139266,-0.491072,0.870802,-0.0234724],[0,-1,-1,0],[9E+09,9E+09,9E+09,9E+09,9E+09,9E+09]],
        [[1366.7,4.5,938.01],[0.00139266,-0.491072,0.870802,-0.0234724],[0,-1,-1,0],[9E+09,9E+09,9E+09,9E+09,9E+09,9E+09]],
        [[1370.7,7.5,938.01],[0.00139266,-0.491072,0.870802,-0.0234724],[0,-1,-1,0],[9E+09,9E+09,9E+09,9E+09,9E+09,9E+09]],
        [[1375.7,12,938.01],[0.00139266,-0.491072,0.870802,-0.0234724],[0,-1,-1,0],[9E+09,9E+09,9E+09,9E+09,9E+09,9E+09]],
        [[1379.7,17,938.01],[0.00139266,-0.491072,0.870802,-0.0234724],[0,-1,-1,0],[9E+09,9E+09,9E+09,9E+09,9E+09,9E+09]],
        [[1382.7,21.5,938.01],[0.00139266,-0.491072,0.870802,-0.0234724],[0,-1,-1,0],[9E+09,9E+09,9E+09,9E+09,9E+09,9E+09]],
        [[1385.7,25.5,938.01],[0.00139266,-0.491072,0.870802,-0.0234724],[0,-1,-1,0],[9E+09,9E+09,9E+09,9E+09,9E+09,9E+09]],
        [[1388.7,29,938.01],[0.00139266,-0.491072,0.870802,-0.0234724],[0,-1,-1,0],[9E+09,9E+09,9E+09,9E+09,9E+09,9E+09]],
        [[1388.2,33,938.01],[0.00139266,-0.491072,0.870802,-0.0234724],[0,-1,-1,0],[9E+09,9E+09,9E+09,9E+09,9E+09,9E+09]],
        [[1387.7,37.5,938.01],[0.00139266,-0.491072,0.870802,-0.0234724],[0,-1,-1,0],[9E+09,9E+09,9E+09,9E+09,9E+09,9E+09]],
        [[1390.7,42,938.01],[0.00139266,-0.491072,0.870802,-0.0234724],[0,-1,-1,0],[9E+09,9E+09,9E+09,9E+09,9E+09,9E+09]],
        [[1395.2,43.5,938.01],[0.00139266,-0.491072,0.870802,-0.0234724],[0,-1,-1,0],[9E+09,9E+09,9E+09,9E+09,9E+09,9E+09]],
        [[1398.2,49,938.01],[0.00139266,-0.491072,0.870802,-0.0234724],[0,-1,-1,0],[9E+09,9E+09,9E+09,9E+09,9E+09,9E+09]],
        [[1398.2,55,938.01],[0.00139266,-0.491072,0.870802,-0.0234724],[0,-1,-1,0],[9E+09,9E+09,9E+09,9E+09,9E+09,9E+09]],
        [[1395.7,59,938.01],[0.00139266,-0.491072,0.870802,-0.0234724],[0,-1,-1,0],[9E+09,9E+09,9E+09,9E+09,9E+09,9E+09]],
        [[1392.7,63.5,938.01],[0.00139266,-0.491072,0.870802,-0.0234724],[0,-1,-1,0],[9E+09,9E+09,9E+09,9E+09,9E+09,9E+09]],
        [[1389.7,67,938.01],[0.00139266,-0.491072,0.870802,-0.0234724],[0,-1,-1,0],[9E+09,9E+09,9E+09,9E+09,9E+09,9E+09]],
        [[1385.2,70.5,938.01],[0.00139266,-0.491072,0.870802,-0.0234724],[0,-1,-1,0],[9E+09,9E+09,9E+09,9E+09,9E+09,9E+09]],
        [[1380.7,73.5,938.01],[0.00139266,-0.491072,0.870802,-0.0234724],[0,-1,-1,0],[9E+09,9E+09,9E+09,9E+09,9E+09,9E+09]],
        [[1375.7,75.5,938.01],[0.00139266,-0.491072,0.870802,-0.0234724],[0,-1,-1,0],[9E+09,9E+09,9E+09,9E+09,9E+09,9E+09]],
        [[1371.2,77,938.01],[0.00139266,-0.491072,0.870802,-0.0234724],[0,-1,-1,0],[9E+09,9E+09,9E+09,9E+09,9E+09,9E+09]],
        [[1366.7,78.5,938.01],[0.00139266,-0.491072,0.870802,-0.0234724],[0,-1,-1,0],[9E+09,9E+09,9E+09,9E+09,9E+09,9E+09]],
        [[1361.7,79.5,938.01],[0.00139266,-0.491072,0.870802,-0.0234724],[0,-1,-1,0],[9E+09,9E+09,9E+09,9E+09,9E+09,9E+09]],
        [[1354.2,80.5,938.01],[0.00139266,-0.491072,0.870802,-0.0234724],[0,-1,-1,0],[9E+09,9E+09,9E+09,9E+09,9E+09,9E+09]],
        [[1344.2,80.5,938.01],[0.00139266,-0.491072,0.870802,-0.0234724],[0,-1,-1,0],[9E+09,9E+09,9E+09,9E+09,9E+09,9E+09]],
        [[1338.7,79.5,938.01],[0.00139266,-0.491072,0.870802,-0.0234724],[0,-1,-1,0],[9E+09,9E+09,9E+09,9E+09,9E+09,9E+09]],
        [[1334.2,77.5,938.01],[0.00139266,-0.491072,0.870802,-0.0234724],[0,-1,-1,0],[9E+09,9E+09,9E+09,9E+09,9E+09,9E+09]],
        [[1328.7,74.5,938.01],[0.00139266,-0.491072,0.870802,-0.0234724],[0,-1,-1,0],[9E+09,9E+09,9E+09,9E+09,9E+09,9E+09]],
        [[1324.2,70.5,938.01],[0.00139266,-0.491072,0.870802,-0.0234724],[0,-1,-1,0],[9E+09,9E+09,9E+09,9E+09,9E+09,9E+09]],
        [[1327.7,67,938.01],[0.00139266,-0.491072,0.870802,-0.0234724],[0,-1,-1,0],[9E+09,9E+09,9E+09,9E+09,9E+09,9E+09]],
        [[1331.7,63,938.01],[0.00139266,-0.491072,0.870802,-0.0234724],[0,-1,-1,0],[9E+09,9E+09,9E+09,9E+09,9E+09,9E+09]],
        [[1334.2,59,938.01],[0.00139266,-0.491072,0.870802,-0.0234724],[0,-1,-1,0],[9E+09,9E+09,9E+09,9E+09,9E+09,9E+09]],
        [[1336.7,54.5,938.01],[0.00139266,-0.491072,0.870802,-0.0234724],[0,-1,-1,0],[9E+09,9E+09,9E+09,9E+09,9E+09,9E+09]],
        [[1338.2,50,938.01],[0.00139266,-0.491072,0.870802,-0.0234724],[0,-1,-1,0],[9E+09,9E+09,9E+09,9E+09,9E+09,9E+09]],
        [[1340.2,45.5,938.01],[0.00139266,-0.491072,0.870802,-0.0234724],[0,-1,-1,0],[9E+09,9E+09,9E+09,9E+09,9E+09,9E+09]],
        [[1341.2,40.5,938.01],[0.00139266,-0.491072,0.870802,-0.0234724],[0,-1,-1,0],[9E+09,9E+09,9E+09,9E+09,9E+09,9E+09]],
        [[1342.7,35.5,938.01],[0.00139266,-0.491072,0.870802,-0.0234724],[0,-1,-1,0],[9E+09,9E+09,9E+09,9E+09,9E+09,9E+09]],
        [[1343.7,30.5,938.01],[0.00139266,-0.491072,0.870802,-0.0234724],[0,-1,-1,0],[9E+09,9E+09,9E+09,9E+09,9E+09,9E+09]],
        [[1344.7,25,938.01],[0.00139266,-0.491072,0.870802,-0.0234724],[0,-1,-1,0],[9E+09,9E+09,9E+09,9E+09,9E+09,9E+09]],
        [[1345.7,19,938.01],[0.00139266,-0.491072,0.870802,-0.0234724],[0,-1,-1,0],[9E+09,9E+09,9E+09,9E+09,9E+09,9E+09]],
        [[1346.2,13,938.01],[0.00139266,-0.491072,0.870802,-0.0234724],[0,-1,-1,0],[9E+09,9E+09,9E+09,9E+09,9E+09,9E+09]],
        [[1344.7,8.5,938.01],[0.00139266,-0.491072,0.870802,-0.0234724],[0,-1,-1,0],[9E+09,9E+09,9E+09,9E+09,9E+09,9E+09]],
        [[1344.2,4,938.01],[0.00139266,-0.491072,0.870802,-0.0234724],[0,-1,-1,0],[9E+09,9E+09,9E+09,9E+09,9E+09,9E+09]],
        [[1348.7,2,938.01],[0.00139266,-0.491072,0.870802,-0.0234724],[0,-1,-1,0],[9E+09,9E+09,9E+09,9E+09,9E+09,9E+09]]
        ];
    CONST robtarget myPath9{7} := [
        [[1360.2,64,938.01],[0.00139266,-0.491072,0.870802,-0.0234724],[0,-1,-1,0],[9E+09,9E+09,9E+09,9E+09,9E+09,9E+09]],
        [[1361.7,69.5,938.01],[0.00139266,-0.491072,0.870802,-0.0234724],[0,-1,-1,0],[9E+09,9E+09,9E+09,9E+09,9E+09,9E+09]],
        [[1367.2,71,938.01],[0.00139266,-0.491072,0.870802,-0.0234724],[0,-1,-1,0],[9E+09,9E+09,9E+09,9E+09,9E+09,9E+09]],
        [[1369.7,67,938.01],[0.00139266,-0.491072,0.870802,-0.0234724],[0,-1,-1,0],[9E+09,9E+09,9E+09,9E+09,9E+09,9E+09]],
        [[1367.2,71,938.01],[0.00139266,-0.491072,0.870802,-0.0234724],[0,-1,-1,0],[9E+09,9E+09,9E+09,9E+09,9E+09,9E+09]],
        [[1361.7,69.5,938.01],[0.00139266,-0.491072,0.870802,-0.0234724],[0,-1,-1,0],[9E+09,9E+09,9E+09,9E+09,9E+09,9E+09]],
        [[1362.2,64,938.01],[0.00139266,-0.491072,0.870802,-0.0234724],[0,-1,-1,0],[9E+09,9E+09,9E+09,9E+09,9E+09,9E+09]]
        ];
    CONST robtarget myPath10{8} := [
        [[1363.2,27.5,938.01],[0.00139266,-0.491072,0.870802,-0.0234724],[0,-1,-1,0],[9E+09,9E+09,9E+09,9E+09,9E+09,9E+09]],
        [[1357.2,31.5,938.01],[0.00139266,-0.491072,0.870802,-0.0234724],[0,-1,-1,0],[9E+09,9E+09,9E+09,9E+09,9E+09,9E+09]],
        [[1355.7,36.5,938.01],[0.00139266,-0.491072,0.870802,-0.0234724],[0,-1,-1,0],[9E+09,9E+09,9E+09,9E+09,9E+09,9E+09]],
        [[1358.7,40.5,938.01],[0.00139266,-0.491072,0.870802,-0.0234724],[0,-1,-1,0],[9E+09,9E+09,9E+09,9E+09,9E+09,9E+09]],
        [[1366.7,41.5,938.01],[0.00139266,-0.491072,0.870802,-0.0234724],[0,-1,-1,0],[9E+09,9E+09,9E+09,9E+09,9E+09,9E+09]],
        [[1371.2,39,938.01],[0.00139266,-0.491072,0.870802,-0.0234724],[0,-1,-1,0],[9E+09,9E+09,9E+09,9E+09,9E+09,9E+09]],
        [[1371.7,34,938.01],[0.00139266,-0.491072,0.870802,-0.0234724],[0,-1,-1,0],[9E+09,9E+09,9E+09,9E+09,9E+09,9E+09]],
        [[1366.7,28,938.01],[0.00139266,-0.491072,0.870802,-0.0234724],[0,-1,-1,0],[9E+09,9E+09,9E+09,9E+09,9E+09,9E+09]]
        ];
    CONST robtarget myPath11{7} := [
        [[1368.2,30.5,938.01],[0.00139266,-0.491072,0.870802,-0.0234724],[0,-1,-1,0],[9E+09,9E+09,9E+09,9E+09,9E+09,9E+09]],
        [[1371.7,33,938.01],[0.00139266,-0.491072,0.870802,-0.0234724],[0,-1,-1,0],[9E+09,9E+09,9E+09,9E+09,9E+09,9E+09]],
        [[1371.7,38,938.01],[0.00139266,-0.491072,0.870802,-0.0234724],[0,-1,-1,0],[9E+09,9E+09,9E+09,9E+09,9E+09,9E+09]],
        [[1367.2,41,938.01],[0.00139266,-0.491072,0.870802,-0.0234724],[0,-1,-1,0],[9E+09,9E+09,9E+09,9E+09,9E+09,9E+09]],
        [[1362.2,41.5,938.01],[0.00139266,-0.491072,0.870802,-0.0234724],[0,-1,-1,0],[9E+09,9E+09,9E+09,9E+09,9E+09,9E+09]],
        [[1361.2,36,938.01],[0.00139266,-0.491072,0.870802,-0.0234724],[0,-1,-1,0],[9E+09,9E+09,9E+09,9E+09,9E+09,9E+09]],
        [[1364.2,32,938.01],[0.00139266,-0.491072,0.870802,-0.0234724],[0,-1,-1,0],[9E+09,9E+09,9E+09,9E+09,9E+09,9E+09]]
        ];
    CONST robtarget myPath12{8} := [
        [[1362.7,28,938.01],[0.00139266,-0.491072,0.870802,-0.0234724],[0,-1,-1,0],[9E+09,9E+09,9E+09,9E+09,9E+09,9E+09]],
        [[1368.2,29.5,938.01],[0.00139266,-0.491072,0.870802,-0.0234724],[0,-1,-1,0],[9E+09,9E+09,9E+09,9E+09,9E+09,9E+09]],
        [[1364.2,32,938.01],[0.00139266,-0.491072,0.870802,-0.0234724],[0,-1,-1,0],[9E+09,9E+09,9E+09,9E+09,9E+09,9E+09]],
        [[1361.2,35.5,938.01],[0.00139266,-0.491072,0.870802,-0.0234724],[0,-1,-1,0],[9E+09,9E+09,9E+09,9E+09,9E+09,9E+09]],
        [[1361.7,41,938.01],[0.00139266,-0.491072,0.870802,-0.0234724],[0,-1,-1,0],[9E+09,9E+09,9E+09,9E+09,9E+09,9E+09]],
        [[1356.7,38.5,938.01],[0.00139266,-0.491072,0.870802,-0.0234724],[0,-1,-1,0],[9E+09,9E+09,9E+09,9E+09,9E+09,9E+09]],
        [[1356.2,33.5,938.01],[0.00139266,-0.491072,0.870802,-0.0234724],[0,-1,-1,0],[9E+09,9E+09,9E+09,9E+09,9E+09,9E+09]],
        [[1359.7,29,938.01],[0.00139266,-0.491072,0.870802,-0.0234724],[0,-1,-1,0],[9E+09,9E+09,9E+09,9E+09,9E+09,9E+09]]
        ];

    PROC draw_path0()
        SetDO SETPEN, 0;
        MoveL myPath0{1}, v50, z5, AW_Gun;
        WaitTime 1;
        SetDO SETPEN, 1;
        FOR i FROM 2 TO Dim(myPath0, 1) DO
            MoveL myPath0{i}, v50, z5, AW_Gun;
        ENDFOR
        WaitTime 0.5;
    ENDPROC
    PROC draw_path1()
        SetDO SETPEN, 0;
        MoveL myPath1{1}, v50, z5, AW_Gun;
        WaitTime 1;
        SetDO SETPEN, 1;
        FOR i FROM 2 TO Dim(myPath1, 1) DO
            MoveL myPath1{i}, v50, z5, AW_Gun;
        ENDFOR
        WaitTime 0.5;
    ENDPROC
    PROC draw_path2()
        SetDO SETPEN, 0;
        MoveL myPath2{1}, v50, z5, AW_Gun;
        WaitTime 1;
        SetDO SETPEN, 1;
        FOR i FROM 2 TO Dim(myPath2, 1) DO
            MoveL myPath2{i}, v50, z5, AW_Gun;
        ENDFOR
        WaitTime 0.5;
    ENDPROC
    PROC draw_path3()
        SetDO SETPEN, 0;
        MoveL myPath3{1}, v50, z5, AW_Gun;
        WaitTime 1;
        SetDO SETPEN, 1;
        FOR i FROM 2 TO Dim(myPath3, 1) DO
            MoveL myPath3{i}, v50, z5, AW_Gun;
        ENDFOR
        WaitTime 0.5;
    ENDPROC
    PROC draw_path4()
        SetDO SETPEN, 0;
        MoveL myPath4{1}, v50, z5, AW_Gun;
        WaitTime 1;
        SetDO SETPEN, 1;
        FOR i FROM 2 TO Dim(myPath4, 1) DO
            MoveL myPath4{i}, v50, z5, AW_Gun;
        ENDFOR
        WaitTime 0.5;
    ENDPROC
    PROC draw_path5()
        SetDO SETPEN, 0;
        MoveL myPath5{1}, v50, z5, AW_Gun;
        WaitTime 1;
        SetDO SETPEN, 1;
        FOR i FROM 2 TO Dim(myPath5, 1) DO
            MoveL myPath5{i}, v50, z5, AW_Gun;
        ENDFOR
        WaitTime 0.5;
    ENDPROC
    PROC draw_path6()
        SetDO SETPEN, 0;
        MoveL myPath6{1}, v50, z5, AW_Gun;
        WaitTime 1;
        SetDO SETPEN, 1;
        FOR i FROM 2 TO Dim(myPath6, 1) DO
            MoveL myPath6{i}, v50, z5, AW_Gun;
        ENDFOR
        WaitTime 0.5;
    ENDPROC
    PROC draw_path7()
        SetDO SETPEN, 0;
        MoveL myPath7{1}, v50, z5, AW_Gun;
        WaitTime 1;
        SetDO SETPEN, 1;
        FOR i FROM 2 TO Dim(myPath7, 1) DO
            MoveL myPath7{i}, v50, z5, AW_Gun;
        ENDFOR
        WaitTime 0.5;
    ENDPROC
    PROC draw_path8()
        SetDO SETPEN, 0;
        MoveL myPath8{1}, v50, z5, AW_Gun;
        WaitTime 1;
        SetDO SETPEN, 1;
        FOR i FROM 2 TO Dim(myPath8, 1) DO
            MoveL myPath8{i}, v50, z5, AW_Gun;
        ENDFOR
        WaitTime 0.5;
    ENDPROC
    PROC draw_path9()
        SetDO SETPEN, 0;
        MoveL myPath9{1}, v50, z5, AW_Gun;
        WaitTime 1;
        SetDO SETPEN, 1;
        FOR i FROM 2 TO Dim(myPath9, 1) DO
            MoveL myPath9{i}, v50, z5, AW_Gun;
        ENDFOR
        WaitTime 0.5;
    ENDPROC
    PROC draw_path10()
        SetDO SETPEN, 0;
        MoveL myPath10{1}, v50, z5, AW_Gun;
        WaitTime 1;
        SetDO SETPEN, 1;
        FOR i FROM 2 TO Dim(myPath10, 1) DO
            MoveL myPath10{i}, v50, z5, AW_Gun;
        ENDFOR
        WaitTime 0.5;
    ENDPROC
    PROC draw_path11()
        SetDO SETPEN, 0;
        MoveL myPath11{1}, v50, z5, AW_Gun;
        WaitTime 1;
        SetDO SETPEN, 1;
        FOR i FROM 2 TO Dim(myPath11, 1) DO
            MoveL myPath11{i}, v50, z5, AW_Gun;
        ENDFOR
        WaitTime 0.5;
    ENDPROC
    PROC draw_path12()
        SetDO SETPEN, 0;
        MoveL myPath12{1}, v50, z5, AW_Gun;
        WaitTime 1;
        SetDO SETPEN, 1;
        FOR i FROM 2 TO Dim(myPath12, 1) DO
            MoveL myPath12{i}, v50, z5, AW_Gun;
        ENDFOR
        WaitTime 0.5;
    ENDPROC

    PROC main()
        SetDO SETPEN, 0;
        WaitTime 1;
        draw_path0;
        WaitTime 0.5;
        draw_path1;
        WaitTime 0.5;
        draw_path2;
        WaitTime 0.5;
        draw_path3;
        WaitTime 0.5;
        draw_path4;
        WaitTime 0.5;
        draw_path5;
        WaitTime 0.5;
        draw_path6;
        WaitTime 0.5;
        draw_path7;
        WaitTime 0.5;
        draw_path8;
        WaitTime 0.5;
        draw_path9;
        WaitTime 0.5;
        draw_path10;
        WaitTime 0.5;
        draw_path11;
        WaitTime 0.5;
        draw_path12;
        WaitTime 0.5;
        SetDO SETPEN, 0;
    ENDPROC

ENDMODULE
